FUNCTION_BLOCK AxisPowerTestSuite EXTENDS TestSuite<TestSuiteParameter.MaxTestCount>
VAR
	StubAxis : AXIS_REF;
	StubTask : I_Task;
	TestAxisPower : EnableBehaviour(StubAxis);
END_VAR

DoesAxisAcceptEnable_Test();
RejectEnableWhenEnabled_Test();
RejectDisableWhenDisabled_Test();

METHOD DoesAxisAcceptEnable_Test : BOOL
VAR_INST
	Expected : BOOL := TRUE;
	Actual	 : BOOL;
END_VAR
IF Test(__POUNAME()).ExecuteTest() THEN
	Actual := SUCCEEDED(TestAxisPower.Enable(StubTask));
	TestAxisPower.Disable(StubTask);
	Test(__POUNAME()).AssertEqual(Expected, Actual);
END_IF
END_METHOD

METHOD RejectDisableWhenDisabled_Test : BOOL
VAR_INST
	Expected : HRESULT;
	Actual	 : HRESULT;
END_VAR
IF Test(__POUNAME()).ExecuteTest() THEN
	Expected := s_false;
	Actual := TestAxisPower.Disable(StubTask);
	Test(__POUNAME()).AssertEqual(Expected, Actual);
END_IF
END_METHOD

METHOD RejectEnableWhenEnabled_Test : BOOL
VAR_INST
	Expected : BOOL := TRUE;
	Actual	 : BOOL;
END_VAR
IF Test(__POUNAME()).ExecuteTest() THEN
	TestAxisPower.Enable(StubTask);
	Actual := FAILED(TestAxisPower.Enable(StubTask));
	TestAxisPower.Disable(StubTask);
	Test(__POUNAME()).AssertEqual(Expected, Actual);
END_IF
END_METHOD

END_FUNCTION_BLOCK

(* stored: Version 1.1.0.1
   POU AxisPowerTestSuite: Id {ac2625ce-9cae-4674-bbac-7fb3863ceb8a}, SpecialFunc None
   Method DoesAxisAcceptEnable_Test: Id {fe79904b-ba9b-4299-9251-955ef4cd651f}
   Method RejectDisableWhenDisabled_Test: Id {2c27dff1-a943-4ffc-b0d9-e00a76c5c4af}
   Method RejectEnableWhenEnabled_Test: Id {3a8db93e-7de7-40e7-bc08-d2e3cb8c9735} *)
